FUNCTION_BLOCK FB_FlowUnits_Tests EXTENDS TcUnit.FB_TestSuite
VAR_INPUT
END_VAR
VAR_OUTPUT
END_VAR
VAR
END_VAR

Test_AllFlowUnits();

METHOD Test_AllFlowUnits
VAR_INPUT
END_VAR
TcUnit.TEST('Test_AllFlowUnits');

AssertEquals_STRING('slm', FlowUnits.Slm, 'Returned property value is incorrect.');
AssertEquals_STRING('sccm', FlowUnits.Sccm, 'Returned property value is incorrect.');

TcUnit.TEST_FINISHED();
END_METHOD

END_FUNCTION_BLOCK

(* stored: Version 1.1.0.1, ProductVersion 3.1.4024.14
   POU FB_FlowUnits_Tests: Id {b11eb69e-a31b-039b-05fc-0308d414074b}, SpecialFunc None
   Method Test_AllFlowUnits: Id {8bdbbc76-c7cc-05f9-2340-3fb2be3fcd06} *)
